TYPE ST_ItemPK1_OUT1 :
STRUCT
	Identity		:ST_Identity_PK1_OUT1;
	ItemState		:STRING;
	RejectReason	:ST_RejectReason_PK1_OUT1;
	logs			:ST_logs_PK1_OUT1;
	NoRead			:STRING;
END_STRUCT
END_TYPE

(* stored: Version 1.1.0.1, ProductVersion 3.1.4024.13
   DUT ST_ItemPK1_OUT1: Id {9a14b81b-d6f7-4315-bca9-ed9ab84aeedd} *)
